// TwinCAT 3 PLC project CraneSimulation
// ProgramVersion: 3.1.4023.0
// libraries:
//   Tc2_Standard, * (Beckhoff Automation GmbH)
//   Tc2_System, * (Beckhoff Automation GmbH)
//   Tc3_Module, * (Beckhoff Automation GmbH)
//   VisuSymbols,3.5.10.0,System
// project tree:
//   / GlobalTextList.TcGTLO (not stored), PlcTask.TcTTO, Visualization Manager.TcVMO (not stored)
//   GVLs/ Inputs.TcGVL, Outputs.TcGVL (not stored), Parameters.TcGVL
//   POUs/ CraneSimulation.TcPOU, MAIN.TcPOU (not stored)
//   VISUs/ CraneHMI.TcVIS

CONFIGURATION CraneSimulation
    RESOURCE PLC ON TwinCAT3
        TASK PlcTask(INTERVAL := T#10ms, PRIORITY := 20);
        PROGRAM MAIN WITH PlcTask : MAIN;
    END_RESOURCE
END_CONFIGURATION

// ---- GVLs/Inputs.TcGVL
{attribute 'qualified_only'}
VAR_GLOBAL
	bEnableSimulation : BOOL;
	bStartSimulation : BOOL;
	bAutoMode : BOOL;
	fManualCylinderPositionReference : REAL;
	fCylinderVelocityReference : REAL;
END_VAR

// ---- GVLs/Parameters.TcGVL
{attribute 'qualified_only'}
VAR_GLOBAL
	fCyclicTime : LREAL := 0.01;
	bSimulationRunning : BOOL := FALSE;
END_VAR

// ---- POUs/CraneSimulation.TcPOU
PROGRAM CraneSimulation
VAR
	fInitialVelocity : REAL := 0;
	fInitialPosition : REAL := 0;
END_VAR

IF Inputs.bStartSimulation AND Inputs.bAutoMode THEN
	Outputs.fSimulationTime := Outputs.fSimulationTime + Parameters.fCyclicTime;
ELSE
	Outputs.fSimulationTime := 0;
END_IF

IF Outputs.fSimulationTime > 0 AND Inputs.bAutoMode THEN
	Parameters.bSimulationRunning := TRUE;
ELSE
	Parameters.bSimulationRunning := FALSE;
END_IF

IF Inputs.bAutoMode THEN
	Outputs.fCylinderVelocity := Inputs.fCylinderVelocityReference;
	Outputs.fCylinderPosition := Outputs.fCylinderVelocity * (Outputs.fSimulationTime*Outputs.fSimulationTime)/2 + fInitialVelocity*Outputs.fSimulationTime + fInitialPosition;
ELSE
	Outputs.fCylinderPosition := Inputs.fManualCylinderPositionReference;
END_IF

END_PROGRAM

// ---- VISUs/CraneHMI.TcVIS
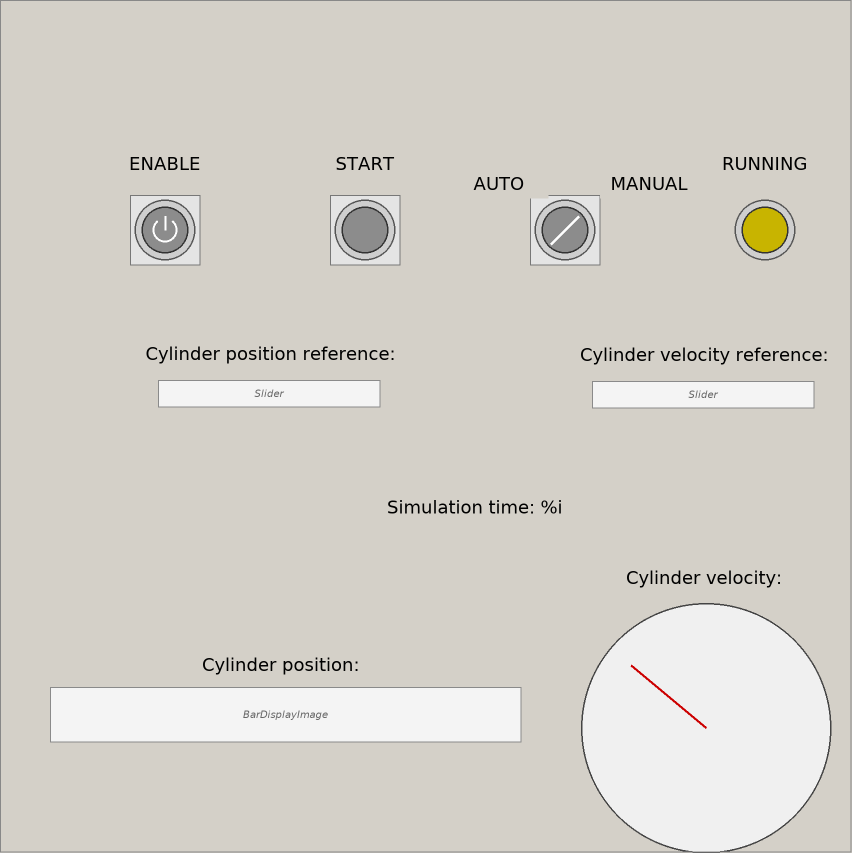
VISUALIZATION CraneHMI  // 852x853
    PowerSwitch (130,195 70x70), variable: Inputs.bEnableSimulation, behaviour: TOGGLE, style: Switch-PowerSwitch-Gray
    RotarySwitch (530,195 70x70), variable: Inputs.bAutoMode, behaviour: TOGGLE, style: Switch-RotarySwitch-Gray
    PushSwitch (330,195 70x70), variable: Inputs.bStartSimulation, behaviour: TOGGLE, style: Switch-PushSwitch-Gray
    Rectangle (115,150 100x28), "ENABLE"
    Rectangle (315,150 100x28), "START"
    Rectangle (450,170 98x28), "AUTO"
    Rectangle (600,170 98x28), "MANUAL"
    Lamp1 (730,195 70x70), variable: Inputs.bEnableSimulation, style: Lamp-Lamp1-Yellow
    Rectangle (715,150 100x28), "RUNNING"
    BarDisplayImage (50,687 471x55), value: Outputs.fCylinderPosition, style: BarDisplayImage-Gray, scale format: %.1f, scale 0..20
    Rectangle (207,494 536x27), "Simulation time: %i", text variable: Outputs.fSimulationTime
    Meter360 (581,603 250x250), value: Outputs.fCylinderVelocity, style: Meter-Meter360-Gray, scale format: %.1f, scale -3..3
    Rectangle (192,652 178x26), "Cylinder position:"
    Rectangle (615,565 178x26), "Cylinder velocity:"
    Slider (158,380 222x27), variable: Inputs.fManualCylinderPositionReference, scale 0..20
    Rectangle (123,342 295x24), "Cylinder position reference:"
    Slider (592,381 222x27), variable: Inputs.fCylinderVelocityReference, scale -3..3
    Rectangle (557,343 295x24), "Cylinder velocity reference:"
END_VISUALIZATION
